RoboDK station: industrial.rdk

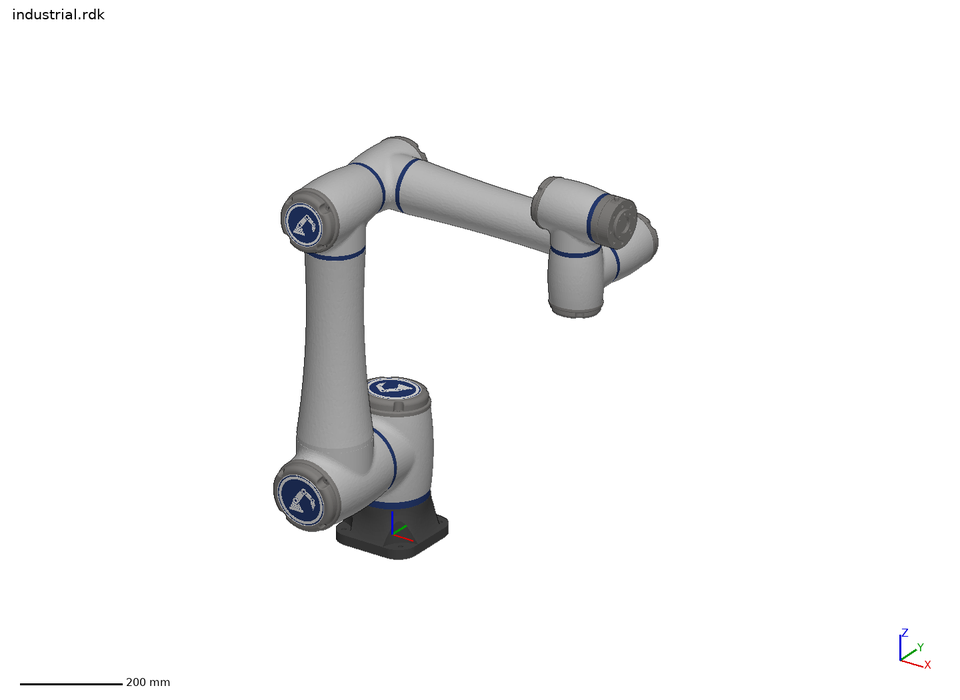
[picture v0: the station drawn from its stored meshes, robots at their saved joint values, targets as dots, program paths as lines]
Station industrial (saved by RoboDK 6.0.1). Poses are relative to the parent item; angles as X-Y-Z fixed-axis rotations.
  - frame RoboDK RDK-COBOT-1200 Base at (0, 0, 0) mm
    - robot RoboDK RDK-COBOT-1200: 6 axes
        modified DH rows (alpha deg, a mm, theta deg, d mm): 0, 0, 0, 201; 90, 0, 90, 0; 0, 590, 0, 0; 0, 560, -90, 175; -90, 0, 0, 140; 90, 0, -90, 117
        joint limits [-360, -180, -160, -180, -180, -360] to [360, 180, 160, 180, 180, 360]; home [0, 0, -90, 90, 90, 0]; saved at [0, 0, -90, 90, 90, 0]
